Staubli VAL3: _getP2PAngle.pgx

public program _getP2PAngle(point x_pHere, point x_pPoint, num& x_nP2PMaxAng[])
  local num l_nResult[14]
begin
  l_nResult[0]=abs(x_pPoint.trsf.rx-x_pHere.trsf.rx)
  l_nResult[1]=abs(x_pPoint.trsf.ry-x_pHere.trsf.ry)
  l_nResult[2]=min(l_nResult[0],360-l_nResult[0])
  l_nResult[3]=min(l_nResult[1],360-l_nResult[1])
  x_nP2PMaxAng=(l_nResult[2]+l_nResult[3])
end
